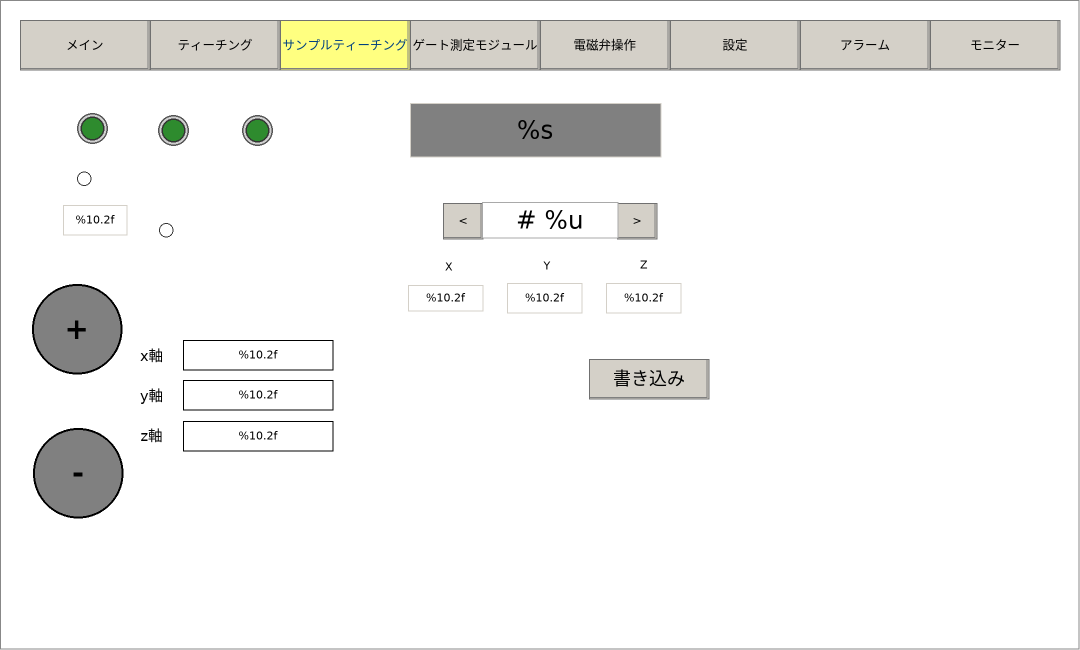
VISUALIZATION s_sample  // 1080x650
    Rectangle (0,0 1080x650)
    Lamp1 (240,113 35x35), variable: gvl_axis.fbi_mc_powerZ.Busy, style: Lamp-Lamp1-Green
    Lamp1 (156,113 35x35), variable: gvl_axis.fbi_mc_powerY.Busy, style: Lamp-Lamp1-Green
    Lamp1 (75,111 35x35), variable: gvl_axis.fbi_mc_powerX.Busy, style: Lamp-Lamp1-Green
    Textfield (63,205 64x30), "%10.2f", text variable: gvl_visu.var_in_inch
        OnMouseClick: write gvl_visu.var_in_inch via VisuDialogs.Numpad, format mm
    Label (126,341 51x30), "x軸"
    Label (126,381 51x30), "y軸"
    Label (126,421 51x30), "z軸"
    Rectangle (183,340 150x30), "%10.2f", text variable: gvl_axis.AxisX.NcToPlc.ActPos
    Rectangle (183,380 150x30), "%10.2f", text variable: gvl_axis.AxisY.NcToPlc.ActPos
    Rectangle (183,421 150x30), "%10.2f", text variable: gvl_axis.AxisZ.NcToPlc.ActPos
    RadioButton (75,159 249x39), variable: gvl_visu.var_jofAxis
    RadioButton (157,210 169x40), variable: gvl_visu.var_radio_jogMode
        Areas[0]: Text=インチ
        Areas[1]: Text=ジョグ
    Ellipse (32,284 90x90), "+", invisible if: gvl_axis.flg_motorReady = FALSE
        OnMouseDown: execute { gvl_visu.flg_btn_moveDirct := eP_direction.positive; }
        OnMouseUp: execute { gvl_visu.flg_btn_moveDirct := eP_direction.keep; }
    Ellipse (33,428 90x90), "-", invisible if: gvl_axis.flg_motorReady = FALSE
        OnMouseDown: execute { gvl_visu.flg_btn_moveDirct := eP_direction.negative; }
        OnMouseUp: execute { gvl_visu.flg_btn_moveDirct := eP_direction.keep; }
    Textfield (408,285 75x26), "%10.2f", text variable: gvl_visu.var_in_samplePos.x
        OnMouseClick: write gvl_visu.var_in_samplePos.x via VisuDialogs.Numpad
    Textfield (507,283 75x30), "%10.2f", text variable: gvl_visu.var_in_samplePos.y
        OnMouseClick: write gvl_visu.var_in_samplePos.y via VisuDialogs.Numpad
    Textfield (606,283 75x30), "%10.2f", text variable: gvl_visu.var_in_samplePos.z
        OnMouseClick: write gvl_visu.var_in_samplePos.z via VisuDialogs.Numpad
    Label (424,252 50x30), "X"
    Label (522,251 50x30), "Y"
    Label (619,250 50x30), "Z"
    Rectangle (410,103 251x54), "%s", text variable: gvl_param.var_productInfo[gvl_param.var_currentProductID].name
    Button (589,359 120x40), "書き込み"
        OnMouseClick: OpenDialog Dialog=d_saveSample, OpenModal=True, OpenCentered=True
    Button (20,20 130x50), "メイン"
        OnMouseClick: change screen: s_auto
    Button (150,20 130x50), "ティーチング"
        OnMouseClick: change screen: s_teaching1
    Button (670,20 130x50), "設定"
        OnMouseClick: change screen: s_setting
    Button (540,20 130x50), "電磁弁操作"
        OnMouseClick: change screen: s_manual
    Button (410,20 130x50), "ゲート測定モジュール"
        OnMouseClick: change screen: s_gm_teaching
    Button (800,20 130x50), "アラーム", colour toggle: gvl_io.flg_signalTowerRed
        OnMouseClick: change screen: s_alarm
    Button (280,20 130x50), "サンプルティーチング"
        OnMouseClick: change screen: s_sample
    Button (617,203 40x36), ">"
        OnMouseClick: execute {
            IF gvl_visu.var_in_sampleCavNo < 8 THEN
            	gvl_visu.var_in_sampleCavNo := gvl_visu.var_in_sampleCavNo + 1;
            END_IF
        }
    Button (443,203 40x36), "<"
        OnMouseClick: execute {
            IF gvl_visu.var_in_sampleCavNo > 1 THEN
            	gvl_visu.var_in_sampleCavNo := gvl_visu.var_in_sampleCavNo - 1;
            END_IF
        }
    Rectangle (482,202 136x36), "# %u", text variable: gvl_visu.var_in_sampleCavNo
    Button (930,20 130x50), "モニター"
        OnMouseClick: change screen: s_monitor
END_VISUALIZATION

(* stored: Version 1.1.0.1, ProductVersion 3.1.4024.11
   Visu s_sample: Id {5fd41c2a-73fe-4e06-954d-ad12d15d60b3} *)
